FUNCTION IntervalIsvalid : BOOL
VAR_INPUT
	pair : REFERENCE TO Interval;
END_VAR

IntervalIsValid := (
	pair.startPos <> GVL.nullPos AND 
	pair.endPos <> GVL.nullPos AND 
	pair.startPos < pair.endPos);

END_FUNCTION

(* stored: Version 1.1.0.1, ProductVersion 3.1.4024.11
   POU IntervalIsvalid: Id {19981972-3874-45d7-bd5a-0c23cbdf8609}, SpecialFunc None *)
